FUNCTION FProcessError : BOOL
VAR_INPUT

///SDOC/////////////////////////////////////////////////////////////////////////
//
//  FProcessError.TcPOU      - Function - PLC error handling - AVT PLC 
//
//  Author:         Mark Colvin                         Date: Sept 5, 2018
//
//	Beckhoff TC3 Structured Text for CX8190 PLC
//
//	includes features:
//		10 inker enables
///////////////////////////////////////////////////////////////////////SDOCEND//

	ErrorNumber :WORD;		//error code to be recorded in the error queue
END_VAR
VAR
	// === LOCAL DATA === NOT saved over power cycles

	Register: WORD;

END_VAR

(************************************************************************************************
 *
 *   FUNCTION 	:FProcessError
 *
 *   Author		:	Mark Colvin
 *
 *   Description:	Place error information into Modbus
 *
 *   Parameters	:	void
 *
 *   Returns	:	void	
 *
 *   History	:   13-Sep-18	MarkC	Created
 *
************************************************************************************************)

// Check if any of the 5 error registers is set to 0 and place error code within it and increment 
//	error count.  If no registry is empty (set to zero) then just add error to error count.
// assume the monitoring slave will read this count and queue array, then zero all values (count & array) in the PLC

GVL.mb_Output_Registers[GVL.ERRORCOUNT]:= GVL.mb_Output_Registers[GVL.ERRORCOUNT] + 1;

FOR Register:= GVL.ERRORREGISTER1 TO GVL.ERRORREGISTER5 DO
	IF (GVL.mb_Output_Registers[Register] = 0) THEN
		GVL.mb_Output_Registers[Register]:= ErrorNumber;
		FProcessError:= TRUE;
		RETURN;
	END_IF
END_FOR
FProcessError:= FALSE;
RETURN;

END_FUNCTION

(* stored: Version 1.1.0.1, ProductVersion 3.1.4022.6
   POU FProcessError: Id {f6606173-48e3-453d-bb25-830548f8a9a2}, SpecialFunc None *)
